// SIMATIC S7-200 project (STEP 7-Micro/WIN), CPU 221 REL 01.10

SYMBOL_TABLE 用户定义1
启动               I0.0
东西灯G             Q0.0
东西灯Y             Q0.1
东西灯R             Q0.2
南北灯G             Q0.3
南北灯Y             Q0.4
南北灯R             Q0.5
END_SYMBOL_TABLE

ORGANIZATION_BLOCK 主程序:OB1
TITLE=程序注释
BEGIN
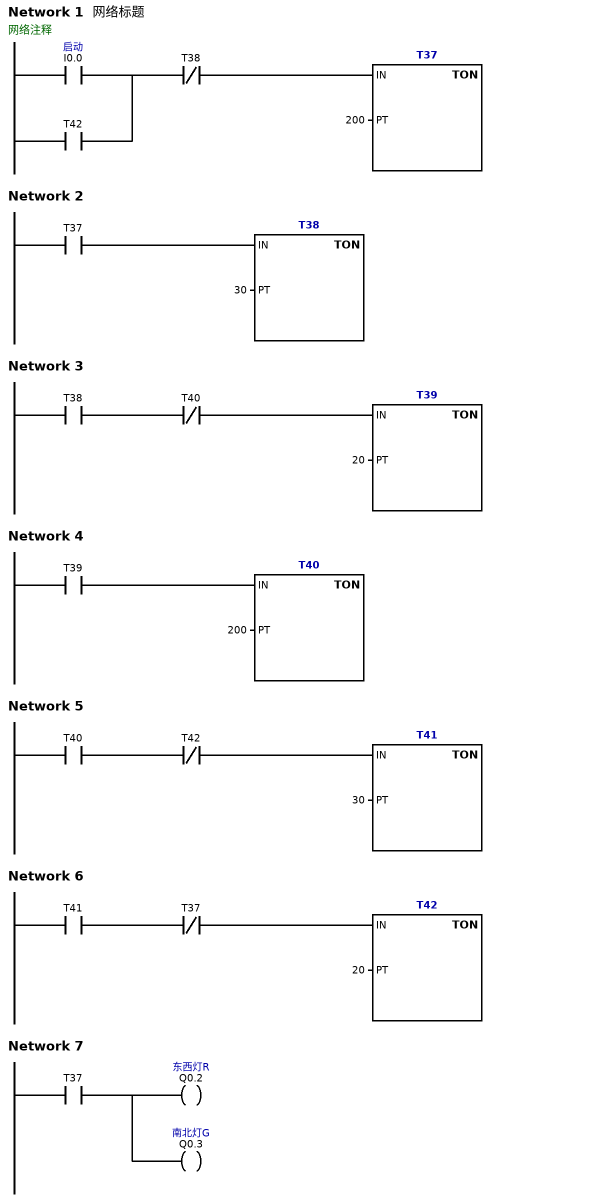
Network 1 // 网络标题
// 网络注释
LD     启动:I0.0
O      T42
AN     T38
TON    T37, 200
Network 2
LD     T37
TON    T38, 30
Network 3
LD     T38
AN     T40
TON    T39, 20
Network 4
LD     T39
TON    T40, 200
Network 5
LD     T40
AN     T42
TON    T41, 30
Network 6
LD     T41
AN     T37
TON    T42, 20
Network 7
LD     T37
=      东西灯R:Q0.2
=      南北灯G:Q0.3
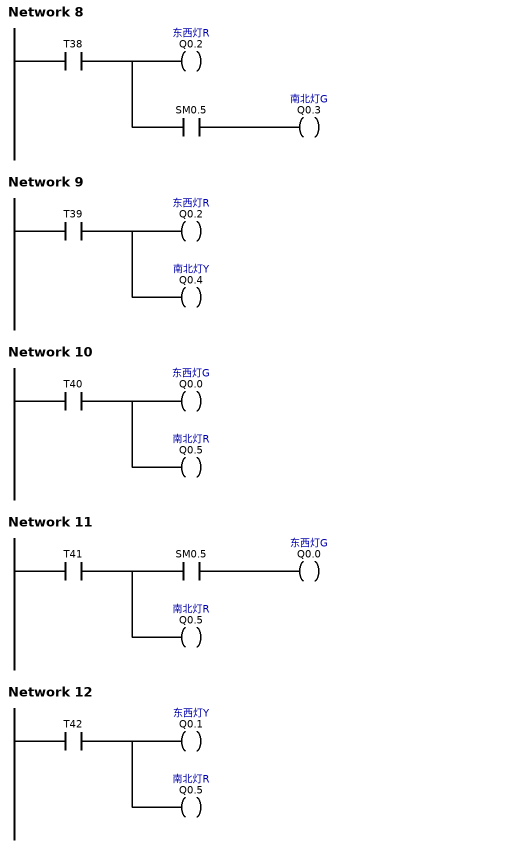
Network 8
LD     T38
=      东西灯R:Q0.2
A      SM0.5
=      南北灯G:Q0.3
Network 9
LD     T39
=      东西灯R:Q0.2
=      南北灯Y:Q0.4
Network 10
LD     T40
=      东西灯G:Q0.0
=      南北灯R:Q0.5
Network 11
LD     T41
LPS
A      SM0.5
=      东西灯G:Q0.0
LPP
=      南北灯R:Q0.5
Network 12
LD     T42
=      东西灯Y:Q0.1
=      南北灯R:Q0.5
END_ORGANIZATION_BLOCK
